PROGRAM MAIN
VAR
END_VAR

END_PROGRAM

(* stored: Version 1.1.0.1, ProductVersion 3.1.0.36
   POU MAIN: Id {f6f8ece3-07cb-43ec-8b46-1b889e76ea23} *)
